ABB RAPID module: DATAROB1.sys

MODULE DATAROB1(SYSMODULE)

    !============================================================================
    !Definition des reperes fixe
    !============================================================================
    !PERS wobjdata Wobj_Table_A:=[FALSE,TRUE,"Table_A",[[-180,-1453.47,766.59],[0.000173821,0.00146815,0.00267763,0.999995]],[[0,0,0],[1,0,0,0]]];
    !PERS wobjdata Wobj_Table_B:=[FALSE,TRUE,"Table_B",[[-179.61,-1453.87,766.37],[0.00106521,0.00081499,0.00296901,0.999995]],[[0,0,0],[1,0,0,0]]];
    PERS wobjdata Wobj_Vision:=[FALSE,TRUE,"",[[-302.07,1699.73,1204.91],[0.00594752,-0.925817,0.377926,2.28926E-05]],[[0,0,0],[1,0,0,0]]];
    !PERS wobjdata Wobj_Vision:=[FALSE,TRUE,"",[[6.64,121.77,1317.72],[0.90213,-0.374443,0.13433,0.167059]],[[0,0,0],[1,0,0,0]]];

    !============================================================================
    !Definition des reperes mobile
    !============================================================================
    PERS wobjdata Wobj_Tool_0:=[TRUE,TRUE,"",[[0,0,0],[1,0,0,0]],[[0,0,0],[1,0,0,0]]];

    PERS wobjdata Wobj_Part_0:=[TRUE,TRUE,"P1",[[0,0,0],[1,0,0,0]],[[0,0,0],[1,0,0,0]]];
    PERS wobjdata Wobj_Part_1:=[TRUE,TRUE,"P1",[[0,0,0],[1,0,0,0]],[[0.155181,-0.746939,-0.01479],[1,-1.91873E-05,-3.53683E-05,-0.000168217]]];
    PERS wobjdata Wobj_Part_2:=[TRUE,TRUE,"P1",[[0,0,0],[1,0,0,0]],[[-0.387538,0.078387,-0.00763113],[1,-1.76602E-05,-7.03178E-07,0.000173258]]];
    PERS wobjdata Wobj_Part_3:=[TRUE,TRUE,"P1",[[0,0,0],[1,0,0,0]],[[-0.030384,-0.00751055,-0.0137897],[1,-8.65311E-06,0.000114207,0.000186753]]];
    PERS wobjdata Wobj_Part_4:=[TRUE,TRUE,"P1",[[0,0,0],[1,0,0,0]],[[-0.682556,0.385389,-0.00285811],[1,3.62591E-05,-1.64536E-05,-0.000709527]]];
    PERS wobjdata Wobj_Part_5:=[TRUE,TRUE,"P1",[[0,0,0],[1,0,0,0]],[[1.0658,-0.0212722,0.210409],[1,9.5615E-06,-0.000719232,-8.11623E-05]]];
    PERS wobjdata Wobj_Part_6:=[TRUE,TRUE,"P1",[[0,0,0],[1,0,0,0]],[[0,0,0],[1,0,0,0]]];
    PERS wobjdata Wobj_Part_7:=[TRUE,TRUE,"P1",[[0,0,0],[1,0,0,0]],[[0,0,0],[1,0,0,0]]];
    PERS wobjdata Wobj_Part_8:=[TRUE,TRUE,"P1",[[0,0,0],[1,0,0,0]],[[0,0,0],[1,0,0,0]]];
    PERS wobjdata Wobj_Part_9:=[TRUE,TRUE,"P1",[[0,0,0],[1,0,0,0]],[[0,0,0],[1,0,0,0]]];

    !======================================
    ! Definition des outils Fixe
    !======================================
    PERS tooldata Tool_Pointe_Fixe:=[FALSE,[[680.531,-1124.32,773.312],[0.707107,2.6E-08,-0.707107,-5E-09]],[150,[3,0,400],[1,0,0,0],4.791,5.093,2.477]];
    PERS tooldata Tool_Mire:=[TRUE,[[-80,140,200],[0.683012702,-0.683012702,-0.183012702,0.183012702]],[150,[3,0,400],[1,0,0,0],4.791,5.093,2.477]];
    PERS tooldata Tool_Pointe:=[TRUE,[[-325.689,-0.27076,55.5616],[0.707032,0.00171379,-0.707178,0.0017141]],[150,[3,0,400],[1,0,0,0],4.791,5.093,2.477]];
    PERS tooldata Tool:=[FALSE,[[1678.28,366.293,1045.02],[0.0132816,-0.00902061,0.70705,-0.706982]],[150,[3,0,400],[1,0,0,0],4.791,5.093,2.477]];
    PERS tooldata Tool_M1:=[FALSE,[[1475.2,610.01,1043.84],[0.50629,0.509351,-0.493533,-0.490568]],[150,[3,0,400],[1,0,0,0],4.791,5.093,2.477]];
    PERS tooldata Tool_M2:=[FALSE,[[1564.3,-813.6,1036.54],[0.502828,0.503332,-0.497149,-0.496652]],[150,[3,0,400],[1,0,0,0],4.791,5.093,2.477]];
    PERS tooldata Tool_M3:=[FALSE,[[1684.22,1216.41,1923.97],[0.503385,0.506672,-0.496526,-0.493304]],[150,[3,0,400],[1,0,0,0],4.791,5.093,2.477]];
    PERS tooldata Tool_M4:=[FALSE,[[1692.3,-1525.57,1929.32],[0.51196,0.509864,-0.48784,-0.489845]],[150,[3,0,400],[1,0,0,0],4.791,5.093,2.477]];
    PERS tooldata Tool_Coin:=[FALSE,[[1606.52,-320.81,971.19],[0.51196,0.509864,-0.48784,-0.489845]],[150,[3,0,400],[1,0,0,0],4.791,5.093,2.477]];


    !---------------------<<<<  LASER  >>>>---------------------
    ! >>> Laser fix
    PERS tooldata Tool_Laser:=[FALSE,[[1832.28,1303.46,1523.26],[0.501194,0.500297,-0.498806,-0.4997]],[150,[3,0,400],[1,0,0,0],4.791,5.093,2.477]];
    !======================================
    ! Definition des outils mobiles
    !======================================
    !Fait le 05/05/2022
    PERS tooldata Tool_Gripper:=[TRUE,[[0,0,380],[1,0,0,0]],[150,[3,0,400],[1,0,0,0],4.791,5.093,2.477]];
    PERS tooldata Tool_Ventouse:=[TRUE,[[0,0,160],[1,0,0,0]],[150,[3,0,400],[1,0,0,0],4.791,5.093,2.477]];
    PERS tooldata Tool_Prehenseur_1:=[TRUE,[[0,0,0],[1,0,0,0]],[150,[3,0,400],[1,0,0,0],4.791,5.093,2.477]];

    !======================================
    ! Definition outils et repères temporaire
    !======================================
    PERS wobjdata Wobj_Table:=[FALSE,TRUE,"Table_B",[[-179.61,-1453.87,766.37],[0.00106521,0.00081499,0.00296901,0.999995]],[[0,0,0],[1,0,0,0]]];

    !============================================================================
    !---------------------<<<<        TABLE WOBJ       >>>>----------------------
    PERS wobjdata wobj_Table_A:=[FALSE,TRUE,"Table_A",[[21.0191,2042.78,502.87],[0.999965,0.000360085,0.00115345,-0.00824105]],[[0,0,0],[1,0,0,0]]];
    PERS wobjdata wobj_Table_B:=[FALSE,TRUE,"Table_B",[[21.3293,2041.93,502.92],[0.999967,0.000148837,0.00134387,-0.00804986]],[[0,0,0],[1,0,0,0]]];

    PERS tooldata ToolCurrent:=[TRUE,[[0,0,0],[1,0,0,0]],[0.001,[0,0,0.001],[1,0,0,0],0,0,0]];
    PERS wobjdata WobjCurrent:=[FALSE,TRUE,"",[[0,0,0],[1,0,0,0]],[[0,0,0],[1,0,0,0]]];

    !======================================
    ! Position specifique  (Robtarget)
    !======================================
    CONST jointtarget P_PEO:=[[90,-60,18,0,90,0],[9E+09,9E+09,9E+09,9E+09,9E+09,9E+09]];
    CONST jointtarget P_REPLI:=[[90,-60,18,0,90,-300],[9E+09,9E+09,9E+09,9E+09,9E+09,9E+09]];

    !Dégagement / Approche Table chargement
    !CONST jointtarget P_App_Table:=[[-96.1806,-32.5627,22.32,0.00020917,58.0012,-0.000940905],[9E+09,9E+09,9E+09,9E+09,9E+09,9E+09]];

    !Point Prise / Dépose
    !PERS robtarget P_Prise_Depose:=[[226.86,218.87,24.2],[0.00037461,-0.368653,-0.929567,-0.000841778],[-2,0,1,0],[9E+09,9E+09,9E+09,9E+09,9E+09,9E+09]];

    !Dégagement / Approche Mur outil 1 et 2
    !CONST jointtarget P_MOTOR_1_2:=[[-3.17104,-35.2057,28.623,12.0352,42.2976,-14.8319],[9E+09,9E+09,9E+09,9E+09,9E+09,9E+09]];
    !Dégagement / Approche Mur outil 3 et 4
    !CONST jointtarget P_MOTOR_3_4:=[[27.3568,-25.5876,27.7485,62.9636,68.9047,-82.1416],[9E+09,9E+09,9E+09,9E+09,9E+09,9E+09]];

    !=========================
    ! Definition zones
    !=========================
    VAR wzstationary wz_REPLI;
    VAR wzstationary wz_PEO;
    VAR shapedata zone_REPLI;
    VAR shapedata zone_PEO;
    !Delta of 2° by joint
    CONST jointtarget DeltaWz:=[[2,2,2,2,2,2],[9E+09,9E+09,9E+09,9E+09,9E+09,9E+09]];

    !=========================
    ! Numeric/bool
    !=========================
    PERS num Code;
    PERS num NumPiece;

    !=========================
    !Declaration des vitesses (speed) / Zones (ZoneData)
    !=========================
    ! Global Speed
    PERS speeddata V_Very_Slow:=[10,5,500,50];
    PERS speeddata V_Slow:=[20,40,500,50];
    PERS speeddata V_Average:=[700,200,500,50];
    PERS speeddata V_Fast:=[1000,500,500,50];
    PERS speeddata V_very_fast:=[1500,400,500,50];

    !Sawing speed
    PERS speeddata V_Sawing_Very_Slow:=[3,5,10,50];
    PERS speeddata V_Sawing_Slow:=[5,10,10,50];
    PERS speeddata V_Sawing:=[10,15,10,50];
    PERS speeddata V_Sawing_Fast:=[15,30,10,50];
    PERS speeddata V_Sawing_Very_Fast:=[20,10,500,50];

    !Grinding speed
    PERS speeddata V_Grinding_Very_Slow:=[10,50,500,50];
    PERS speeddata V_Grinding_Slow:=[20,20,500,50];
    PERS speeddata v_Grinding_Average:=[50,70,500,50];
    PERS speeddata V_Grinding:=[35,60,500,50];
    PERS speeddata V_Grinding_Fast:=[70,80,500,50];

    !Drilling speed
    PERS speeddata V_Drilling:=[3,50,500,50];

    !finition speed
    PERS speeddata V_Finition_Slow:=[15,15,500,50];
    PERS speeddata V_Finition_Average:=[40,18,500,50];
    PERS speeddata V_Finition:=[30,30,500,50];
    PERS speeddata V_Finition_Fast:=[50,30,500,50];

ENDMODULE
